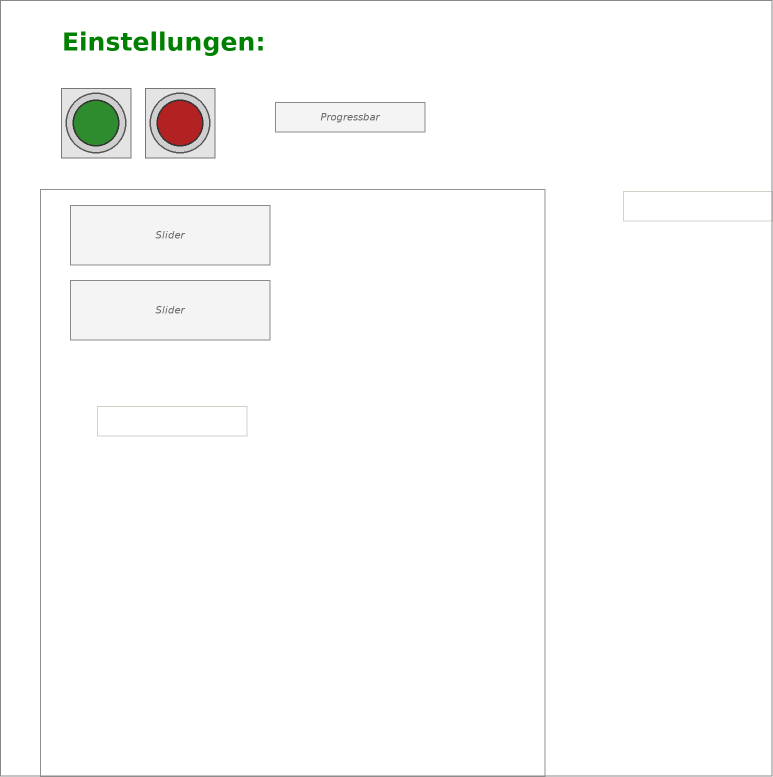
VISUALIZATION Einstellungen  // 773x777
    Label (29,20 270x43), "Einstellungen:"
    PushSwitchLed (145,88 70x70), tooltip "off", variable: MAIN.bOffButtonPressed, behaviour: TOGGLE, style: Switch-PushSwitchLed-Red
    Progressbar (275,102 150x30), variable: MAIN.fbStateMachine.timerTON.ET
    PushSwitchLed (61,88 70x70), tooltip "on", variable: MAIN.bOnButtonPressed, behaviour: TOGGLE, style: Switch-PushSwitchLed-Green
    GroupBox (40,181 505x596)
        Slider (30,24 200x60), variable: GVL.configValues.targetTemperatureOn, scale 20..60
            p2985826283: %i °C
        Slider (30,99 200x60), variable: GVL.configValues.targetTemperatureOff, scale 20..80
            p2985826283: %i °C
        Textfield (57,225 150x30), tooltip "minimale Temperastur am Verdampfer-Ausgangs", text variable: GVL.configValues.evaporatingTemperatureOutMin
    Textfield (623,191 150x30), tooltip "Temperatur Puffer Open", text variable: MAIN.fbProcessdata.pd.sensor.bufferTopTemperature
END_VISUALIZATION

(* stored: Version 1.1.0.1
   Visu Einstellungen: Id {d0de47ec-3ee8-4983-acda-82686d72ed3c} *)
